// TIA Portal V19 export
DATA_BLOCK "Air_Flow_IDB"   // DB185
// stored: InstanceOfName Air_Flow, InstanceOfType FB
"Air_Flow"
   // VAR
   //    AirCounter : Real;
   //    Aux1s : Bool;
   // END_VAR
BEGIN
END_DATA_BLOCK
